{attribute addProperty BoxType "EL9930-0000-0017"}
{attribute addProperty Id "A_0004_EL9930_0001_0017EL9930_AECBF7E8324"}
{attribute addProperty CRC "3116326209"}
{attribute addProperty SizeInBites "32"}
{attribute addProperty SizeInBytes "4"}
TYPE A_0003_EL9930_0000_0017_B9BF5D41 EXTENDS EL9930_D743E87C :
STRUCT
	{attribute addProperty Name "A_0004_EL9930_0001_0017"}
	A_0004_EL9930_0001_0017 : EL9930_AECBF7E8;
END_STRUCT
END_TYPE

(* stored: Version 1.2.0.0, ProductVersion 3.1.4024.9
   DUT A_0003_EL9930_0000_0017_B9BF5D41: Id {bfe54b05-1d56-4539-a257-6a07b74b475b} *)
